FUNCTION_BLOCK logiBUS_8_DI_DOUBLE_CLICK (* Button double click --> IE *)
  (* Function: All Inputs; Description: Copyright (c) 2018, 2023 Jose Cabral, HR Agrartechnik GmbH This program and the accompanying materials are made available under the terms of the Eclipse Public License 2.0 which is available at https://www.eclipse.org/legal/epl-2.0/ SPDX-License-Identifier: EPL-2.0 this maps to IE *)
  (* Version 1.0, 2018-12-05, Jose Cabral *)
  (* Version 1.1, 2022-08-04, Franz Höpfinger, HR Agrartechnik GmbH *)
  (* Version 1.2, 2023-01-05, Franz Höpfinger, HR Agrartechnik GmbH *)
  (* Version 1.3, 2025-02-18, Franz Höpfinger, HR Agrartechnik GmbH, logiBUS IO created. *)
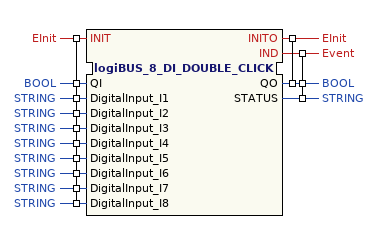
  EVENT_INPUT
    INIT : EInit WITH QI, DigitalInput_I1, DigitalInput_I2, DigitalInput_I3, DigitalInput_I4, DigitalInput_I5, DigitalInput_I6, DigitalInput_I7, DigitalInput_I8; (* Service Initialization *)
  END_EVENT
  EVENT_OUTPUT
    INITO : EInit WITH QO; (* Initialization Confirm *)
    IND WITH QO, STATUS; (* Indication from Resource *)
  END_EVENT
  VAR_INPUT
    QI : BOOL; (* Event Input Qualifier *)
    DigitalInput_I1 : STRING; (* Identifier for Input 1 *)
    DigitalInput_I2 : STRING; (* Identifier for Input 2 *)
    DigitalInput_I3 : STRING; (* Identifier for Input 3 *)
    DigitalInput_I4 : STRING; (* Identifier for Input 4 *)
    DigitalInput_I5 : STRING; (* Identifier for Input 5 *)
    DigitalInput_I6 : STRING; (* Identifier for Input 6 *)
    DigitalInput_I7 : STRING; (* Identifier for Input 7 *)
    DigitalInput_I8 : STRING; (* Identifier for Input 8 *)
  END_VAR
  VAR_OUTPUT
    QO : BOOL; (* Event Output Qualifier *)
    STATUS : STRING; (* Service Status *)
  END_VAR
END_FUNCTION_BLOCK
